// Mitsubishi GX Works2 project: PLC   PLC: FX3G

// global labels: Global1
VAR_GLOBAL
  Start_Day AT X007 : BOOL;
  Emergency_Switch AT X005 : BOOL;
  Work_Day AT Y007 : BOOL;
  Y7coil AT Y007 : BOOL;
  MoveInput AT X007 : BOOL;
  RaspInput AT D1100 : REAL;
  RaspInventory AT D1110 : REAL;
  LemonInput AT D1102 : REAL;
  LemonInventory AT D1112 : REAL;
  StabilizerInput AT D1104 : REAL;
  StabilizerInventory AT D1114 : REAL;
  GummyBearsInput AT D1106 : REAL;
  GummyBearsInventory AT D1116 : REAL;
  ReadyGummyGumPackage AT D1108 : REAL;
  Start_Making AT X001 : BOOL;
  Analog_Input AT D8280 : INT;
  Analog_Float AT D8280 : REAL;
END_VAR
VAR_GLOBAL CONSTANT
  Div400 : REAL := 400;
END_VAR
VAR_GLOBAL
  GummyChoice AT D7000 : REAL;
END_VAR
VAR_GLOBAL CONSTANT
  Plesure : REAL := 6;
END_VAR
VAR_GLOBAL
  Pleasure_Check AT M0 : BOOL;
END_VAR
VAR_GLOBAL CONSTANT
  Regular : REAL := 5;
END_VAR
VAR_GLOBAL
  Regular_Check AT M1 : BOOL;
END_VAR
VAR_GLOBAL CONSTANT
  MinRasp : REAL := 385;
  MinLemon : REAL := 455;
END_VAR
VAR_GLOBAL
  CheckLemonRegular AT M23 : BOOL;
END_VAR
VAR_GLOBAL CONSTANT
  StabilizerMin : REAL := 105;
END_VAR
VAR_GLOBAL
  CheckStabilizerReg AT M24 : BOOL;
END_VAR
VAR_GLOBAL CONSTANT
  GummyBearsMin : REAL := 28;
END_VAR
VAR_GLOBAL
  CheckGummyBearsReg AT M25 : BOOL;
  YesRegularInv AT M16 : BOOL;
END_VAR
VAR_GLOBAL CONSTANT
  MinRaspReg : REAL := 280;
  MinLemonReg : REAL := 455;
  StabilizerMinReg : REAL := 105;
  GummyBearsMinReg : REAL := 28;
  MinRaspPleas : REAL := 385;
END_VAR
VAR_GLOBAL
  CheckRaspPleas AT M26 : BOOL;
END_VAR
VAR_GLOBAL CONSTANT
  MinLemonPleas : REAL := 665;
END_VAR
VAR_GLOBAL
  CheckLemonPleas AT M27 : BOOL;
END_VAR
VAR_GLOBAL CONSTANT
  StabilizerMinPleas : REAL := 210;
END_VAR
VAR_GLOBAL
  CheckStabilizerPleas AT M28 : BOOL;
END_VAR
VAR_GLOBAL CONSTANT
  GummyBearsMinPleas : REAL := 70;
END_VAR
VAR_GLOBAL
  CheckGummyBearsPleas AT M29 : BOOL;
  CheckRaspReg AT M22 : BOOL;
  YesPleasInv AT M17 : BOOL;
  LackMaterials AT M19 : BOOL;
  IceCreamTimer AT TC1 : BOOL;
END_VAR
VAR_GLOBAL CONSTANT
  IceCreamReady : INT := 50;
END_VAR
VAR_GLOBAL
  InMaking AT TS1 : BOOL;
  MakingProcess AT Y000 : BOOL;
  InMakingProcess AT Y000 : BOOL;
  Start_Cooling AT X002 : BOOL;
  EndMaking AT TS1 : BOOL;
  IceCreamCoolingTimer AT TC2 : BOOL;
END_VAR
VAR_GLOBAL CONSTANT
  IceCreamCool : INT := 80;
END_VAR
VAR_GLOBAL
  InCooling AT TS2 : BOOL;
  TempSens AT X003 : BOOL;
  InCoolingProcess AT Y002 : BOOL;
  Below10Degrees AT X003 : BOOL;
  After8Seconds AT TS2 : BOOL;
  FinishCooloing AT M100 : BOOL;
  gsfg AT M120 : BOOL;
  EndCooking AT TS1 : BOOL;
  FlagEndMaking AT M100 : BOOL;
  RaspIceCreamMaking AT D1210 : REAL;
END_VAR
VAR_GLOBAL CONSTANT
  StabilizerRaspPleas : REAL := 70;
  LemonForRaspPleas : REAL := 105;
END_VAR
VAR_GLOBAL
  LemonIceCreamMaking AT D1212 : REAL;
END_VAR
VAR_GLOBAL CONSTANT
  LemonForLemonPleas : REAL := 560;
  StabilizerLemonPleas : REAL := 140;
  LemonForRaspReg : REAL := 35;
  StabilizeForRaspReg : REAL := 35;
  LemonForLemonReg : REAL := 420;
  StabilzerForLemonReg : REAL := 70;
END_VAR
VAR_GLOBAL
  FlagEndCooling AT M101 : BOOL;
  RaspIceCreamCooling AT D1310 : REAL;
  LemonIceCreamCooling AT D1312 : REAL;
  TimeOfFlicker AT TC3 : BOOL;
END_VAR
VAR_GLOBAL CONSTANT
  FlickeringTimeForPleasure : REAL := 50;
  PleasureFlickeringTime : INT := 50;
END_VAR
VAR_GLOBAL
  TimeOfFlickerRegular AT TC4 : BOOL;
  TimeOfFlickePleas AT TC3 : BOOL;
END_VAR
VAR_GLOBAL CONSTANT
  RegularFlickeringTime : INT := 30;
END_VAR
VAR_GLOBAL
  FlickeringPleas AT TS3 : BOOL;
  FlickeringReg AT TS4 : BOOL;
  MixingContainer AT D1410 : REAL;
  FlickeringHelp AT M10 : BOOL;
  FlickeringLight5IsOver AT TS5 : BOOL;
  BlinkingLight1 AT TC5 : BOOL;
  Light5 AT Y005 : BOOL;
  FlickeringLight2 AT TC6 : BOOL;
  FlickeringLight1 AT TC5 : BOOL;
END_VAR
VAR_GLOBAL CONSTANT
  HalfSecondDuration : INT := 5;
END_VAR
VAR_GLOBAL
  Light6 AT Y006 : BOOL;
  FlickeringLight6IsOver AT TS6 : BOOL;
  StartPackPhase AT X004 : BOOL;
  DonePackage AT CS2 : BOOL;
  PackIceCream AT X000 : BOOL;
  EndPleasureFlickering AT TS3 : BOOL;
  EndRegularFlickering AT TS4 : BOOL;
  FlagEndMixing AT M102 : BOOL;
  ConesCounter AT CC1 : BOOL;
END_VAR
VAR_GLOBAL CONSTANT
  Target : INT := 7;
END_VAR
VAR_GLOBAL
  IceCreamCounter AT CC1 : BOOL;
  FinishPackPhase AT CS1 : BOOL;
  IceCreamCurrentCounter AT CN1 : INT;
END_VAR
VAR_GLOBAL CONSTANT
  Min_For_Y4_Light : INT := 1;
  Max_For_Y4_Light : INT := 6;
END_VAR
VAR_GLOBAL
  Light4 AT Y004 : BOOL;
END_VAR
VAR_GLOBAL CONSTANT
  AddPackage : REAL := 1;
END_VAR
VAR_GLOBAL
  ResetDelay AT TC7 : BOOL;
END_VAR
VAR_GLOBAL CONSTANT
  DelayDuration : INT := 10;
END_VAR
VAR_GLOBAL
  ResetDelayOver AT TS7 : BOOL;
  EndDayReset AT M110 : BOOL;
END_VAR
VAR_GLOBAL CONSTANT
  Normalization : REAL := 40;
END_VAR
VAR_GLOBAL
  NormalizedNumberOfPackages AT D1500 : REAL;
  AnalogOutput AT D8282 : INT;
END_VAR
VAR_GLOBAL CONSTANT
  IngredientsForPleasure : REAL := 190;
  IngredientsForRegular : REAL := 124;
END_VAR
VAR_GLOBAL
  EndIteration AT M200 : BOOL;
END_VAR

// task Task_01 (event TRUE, interval 0, priority 31): POU_01

PROGRAM POU_01
VAR
  CheckRaspRegular : BOOL;
END_VAR
(* structured ladder/FBD written out as ST: instructions are called as NAME(EN, inputs, outputs); _pN, _eN, _tN stand for wires *)
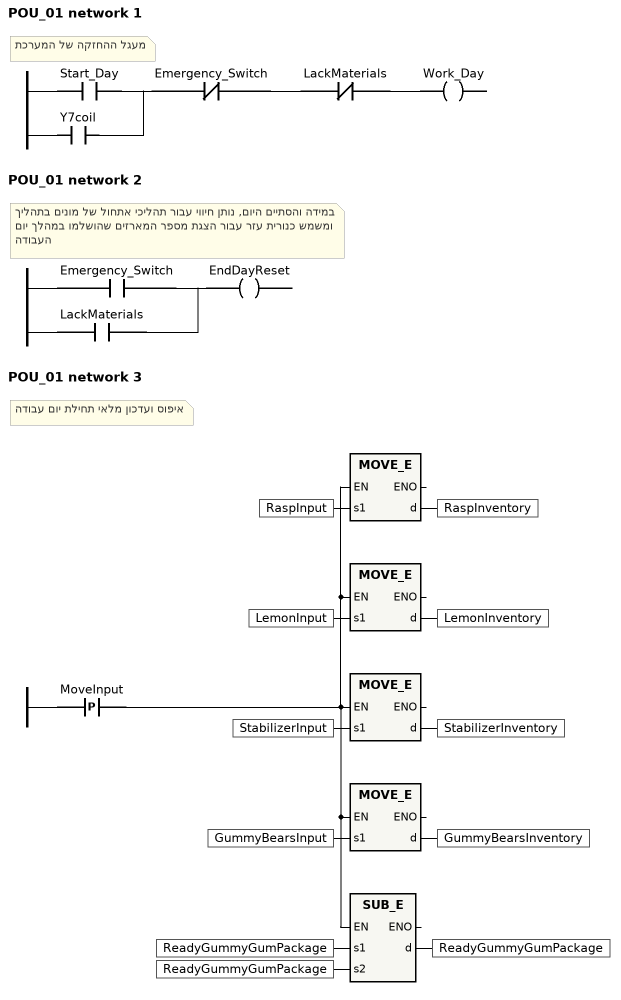
(* network 1 *)
(* מעגל ההחזקה של המערכת *)
Work_Day := ((Start_Day OR Y7coil) AND NOT Emergency_Switch) AND NOT LackMaterials;
(* network 2 *)
(* במידה והסתיים היום, נותן חיווי עבור תהליכי אתחול של מונים בתהליך ומשמש כנורית עזר עבור הצגת מספר המארזים שהושלמו במהלך יום העבודה *)
EndDayReset := Emergency_Switch OR LackMaterials;
(* network 3 *)
(* איפוס ועדכון מלאי תחילת יום עבודה *)
_p1 := LDP(TRUE, MoveInput);
MOVE_E(_p1, RaspInput, RaspInventory);
MOVE_E(_p1, LemonInput, LemonInventory);
MOVE_E(_p1, StabilizerInput, StabilizerInventory);
MOVE_E(_p1, GummyBearsInput, GummyBearsInventory);
SUB_E(_p1, ReadyGummyGumPackage, ReadyGummyGumPackage, ReadyGummyGumPackage);
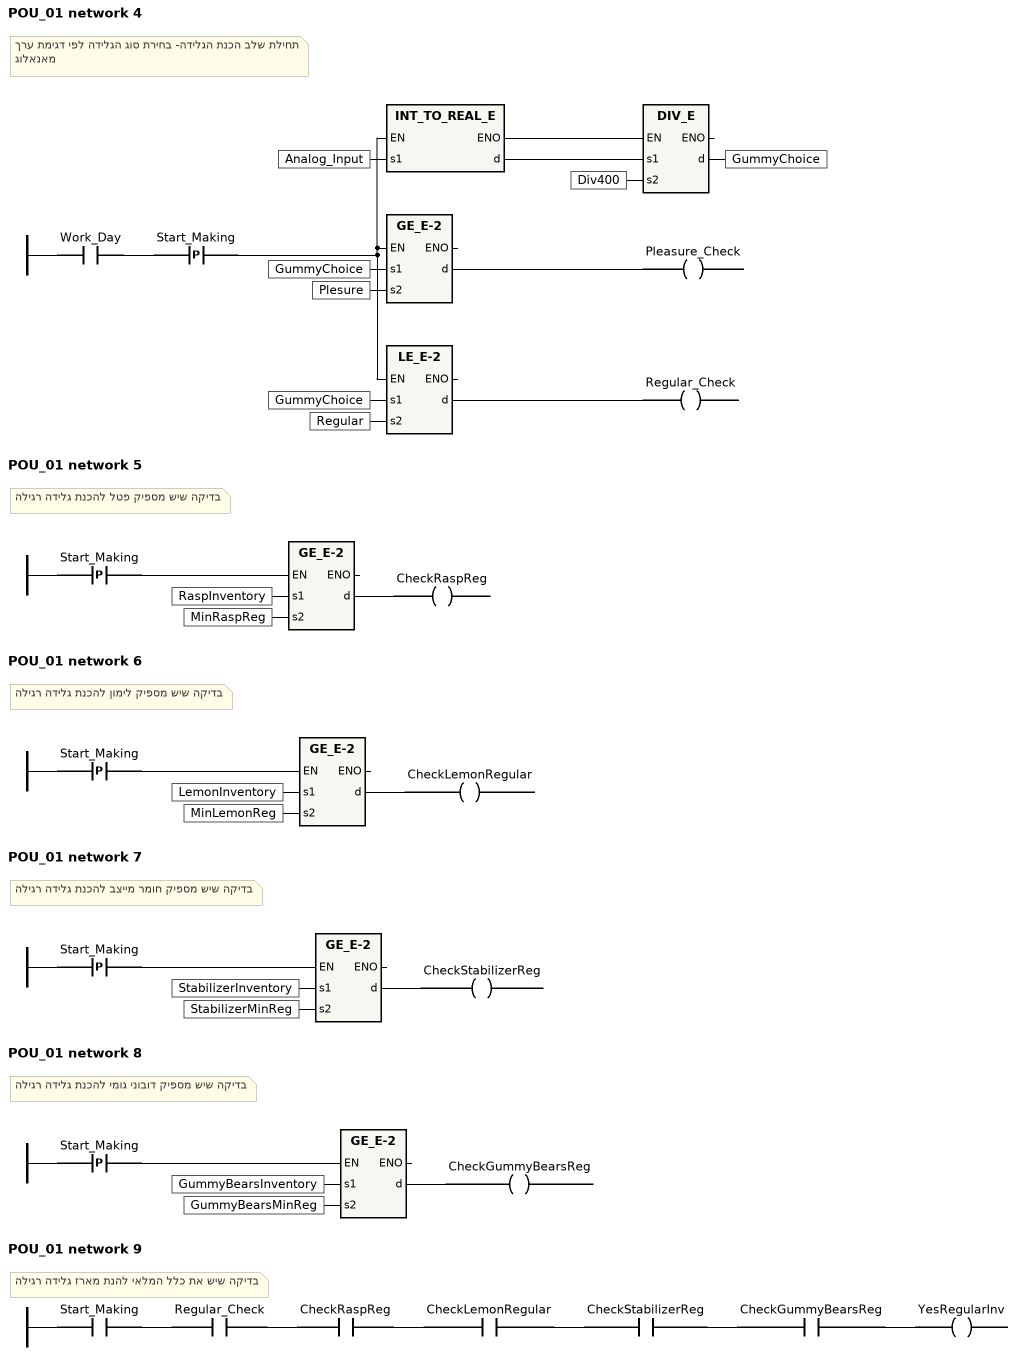
(* network 4 *)
(* תחילת שלב הכנת הגלידה- בחירת סוג הגלידה לפי דגימת ערך מאנאלוג *)
_p1 := Work_Day AND LDP(TRUE, Start_Making);
_e3 := INT_TO_REAL_E(_p1, Analog_Input, _t2);
DIV_E(_e3, _t2, Div400, GummyChoice);
GE_E(_p1, GummyChoice, Plesure, _t4);
Pleasure_Check := _t4;
LE_E(_p1, GummyChoice, Regular, _t5);
Regular_Check := _t5;
(* network 5 *)
(* בדיקה שיש מספיק פטל להכנת גלידה רגילה *)
GE_E(LDP(TRUE, Start_Making), RaspInventory, MinRaspReg, _t1);
CheckRaspReg := _t1;
(* network 6 *)
(* בדיקה שיש מספיק לימון להכנת גלידה רגילה *)
GE_E(LDP(TRUE, Start_Making), LemonInventory, MinLemonReg, _t1);
CheckLemonRegular := _t1;
(* network 7 *)
(* בדיקה שיש מספיק חומר מייצב להכנת גלידה רגילה *)
GE_E(LDP(TRUE, Start_Making), StabilizerInventory, StabilizerMinReg, _t1);
CheckStabilizerReg := _t1;
(* network 8 *)
(* בדיקה שיש מספיק דובוני גומי להכנת גלידה רגילה *)
GE_E(LDP(TRUE, Start_Making), GummyBearsInventory, GummyBearsMinReg, _t1);
CheckGummyBearsReg := _t1;
(* network 9 *)
(* בדיקה שיש את כלל המלאי להנת מארז גלידה רגילה *)
YesRegularInv := Start_Making AND Regular_Check AND CheckRaspReg AND CheckLemonRegular AND CheckStabilizerReg AND CheckGummyBearsReg;
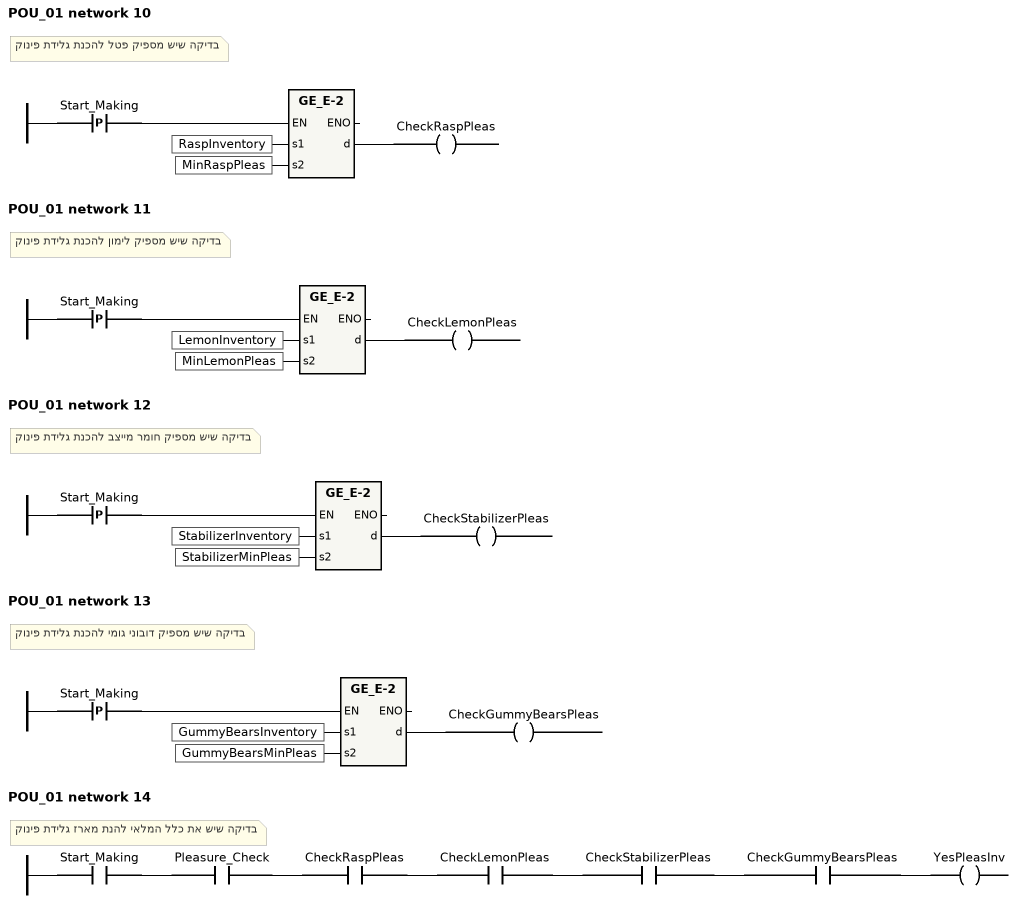
(* network 10 *)
(* בדיקה שיש מספיק פטל להכנת גלידת פינוק *)
GE_E(LDP(TRUE, Start_Making), RaspInventory, MinRaspPleas, _t1);
CheckRaspPleas := _t1;
(* network 11 *)
(* בדיקה שיש מספיק לימון להכנת גלידת פינוק *)
GE_E(LDP(TRUE, Start_Making), LemonInventory, MinLemonPleas, _t1);
CheckLemonPleas := _t1;
(* network 12 *)
(* בדיקה שיש מספיק חומר מייצב להכנת גלידת פינוק *)
GE_E(LDP(TRUE, Start_Making), StabilizerInventory, StabilizerMinPleas, _t1);
CheckStabilizerPleas := _t1;
(* network 13 *)
(* בדיקה שיש מספיק דובוני גומי להכנת גלידת פינוק *)
GE_E(LDP(TRUE, Start_Making), GummyBearsInventory, GummyBearsMinPleas, _t1);
CheckGummyBearsPleas := _t1;
(* network 14 *)
(* בדיקה שיש את כלל המלאי להנת מארז גלידת פינוק *)
YesPleasInv := Start_Making AND Pleasure_Check AND CheckRaspPleas AND CheckLemonPleas AND CheckStabilizerPleas AND CheckGummyBearsPleas;
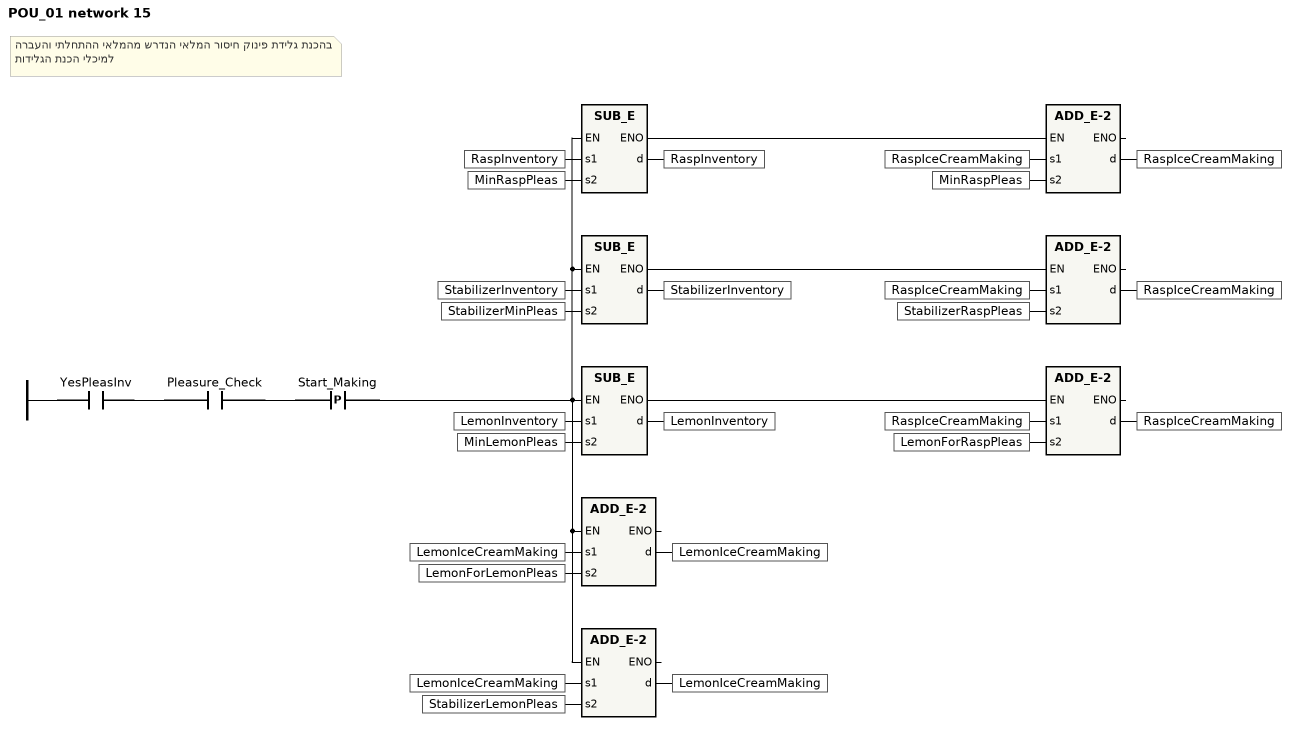
(* network 15 *)
(* בהכנת גלידת פינוק חיסור המלאי הנדרש מהמלאי ההתחלתי והעברה למיכלי הכנת הגלידות *)
_p1 := YesPleasInv AND Pleasure_Check AND LDP(TRUE, Start_Making);
_e2 := SUB_E(_p1, RaspInventory, MinRaspPleas, RaspInventory);
ADD_E(_e2, RaspIceCreamMaking, MinRaspPleas, RaspIceCreamMaking);
_e3 := SUB_E(_p1, StabilizerInventory, StabilizerMinPleas, StabilizerInventory);
ADD_E(_e3, RaspIceCreamMaking, StabilizerRaspPleas, RaspIceCreamMaking);
_e4 := SUB_E(_p1, LemonInventory, MinLemonPleas, LemonInventory);
ADD_E(_e4, RaspIceCreamMaking, LemonForRaspPleas, RaspIceCreamMaking);
ADD_E(_p1, LemonIceCreamMaking, LemonForLemonPleas, LemonIceCreamMaking);
ADD_E(_p1, LemonIceCreamMaking, StabilizerLemonPleas, LemonIceCreamMaking);
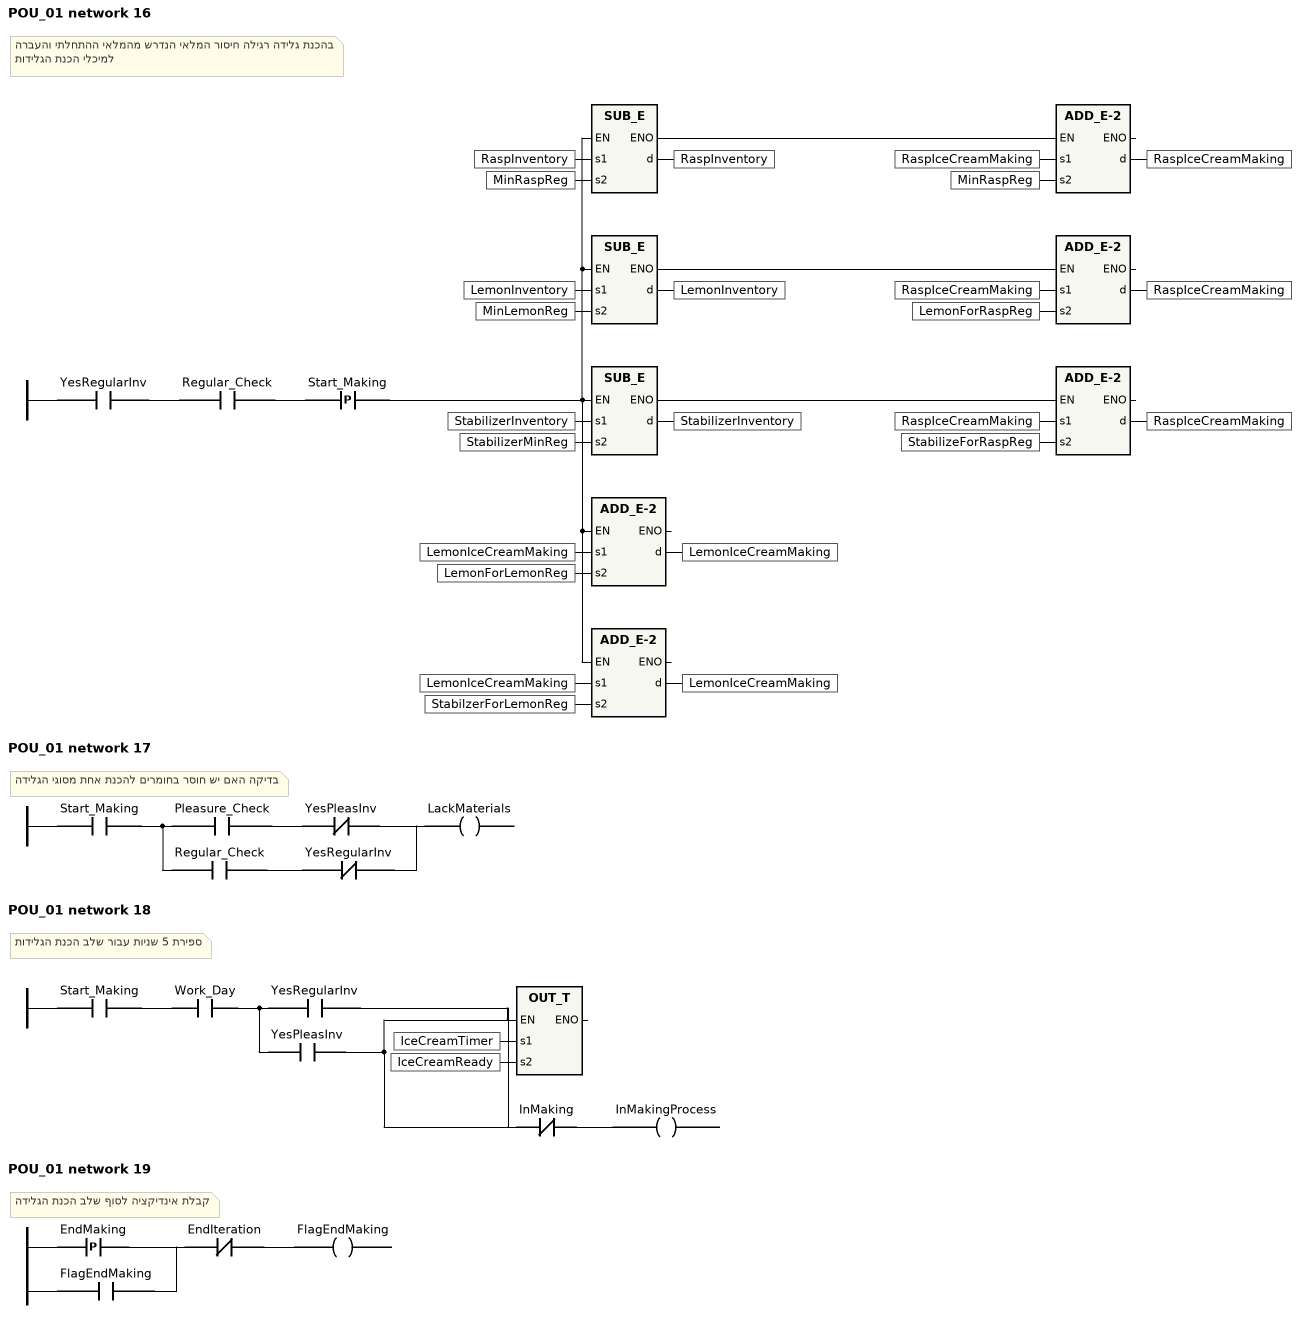
(* network 16 *)
(* בהכנת גלידה רגילה חיסור המלאי הנדרש מהמלאי ההתחלתי והעברה למיכלי הכנת הגלידות *)
_p1 := YesRegularInv AND Regular_Check AND LDP(TRUE, Start_Making);
_e2 := SUB_E(_p1, RaspInventory, MinRaspReg, RaspInventory);
ADD_E(_e2, RaspIceCreamMaking, MinRaspReg, RaspIceCreamMaking);
_e3 := SUB_E(_p1, LemonInventory, MinLemonReg, LemonInventory);
ADD_E(_e3, RaspIceCreamMaking, LemonForRaspReg, RaspIceCreamMaking);
_e4 := SUB_E(_p1, StabilizerInventory, StabilizerMinReg, StabilizerInventory);
ADD_E(_e4, RaspIceCreamMaking, StabilizeForRaspReg, RaspIceCreamMaking);
ADD_E(_p1, LemonIceCreamMaking, LemonForLemonReg, LemonIceCreamMaking);
ADD_E(_p1, LemonIceCreamMaking, StabilzerForLemonReg, LemonIceCreamMaking);
(* network 17 *)
(* בדיקה האם יש חוסר בחומרים להכנת אחת מסוגי הגלידה *)
LackMaterials := (Start_Making AND Pleasure_Check AND NOT YesPleasInv) OR (Start_Making AND Regular_Check AND NOT YesRegularInv);
(* network 18 *)
(* ספירת 5 שניות עבור שלב הכנת הגלידות *)
_p1 := Start_Making AND Work_Day;
_p2 := (_p1 AND YesRegularInv) OR (_p1 AND YesPleasInv);
InMakingProcess := _p2 AND NOT InMaking;
OUT_T(_p2, IceCreamTimer, IceCreamReady);
(* network 19 *)
(* קבלת אינדיקציה לסוף שלב הכנת הגלידה *)
FlagEndMaking := (LDP(TRUE, EndMaking) OR FlagEndMaking) AND NOT EndIteration;
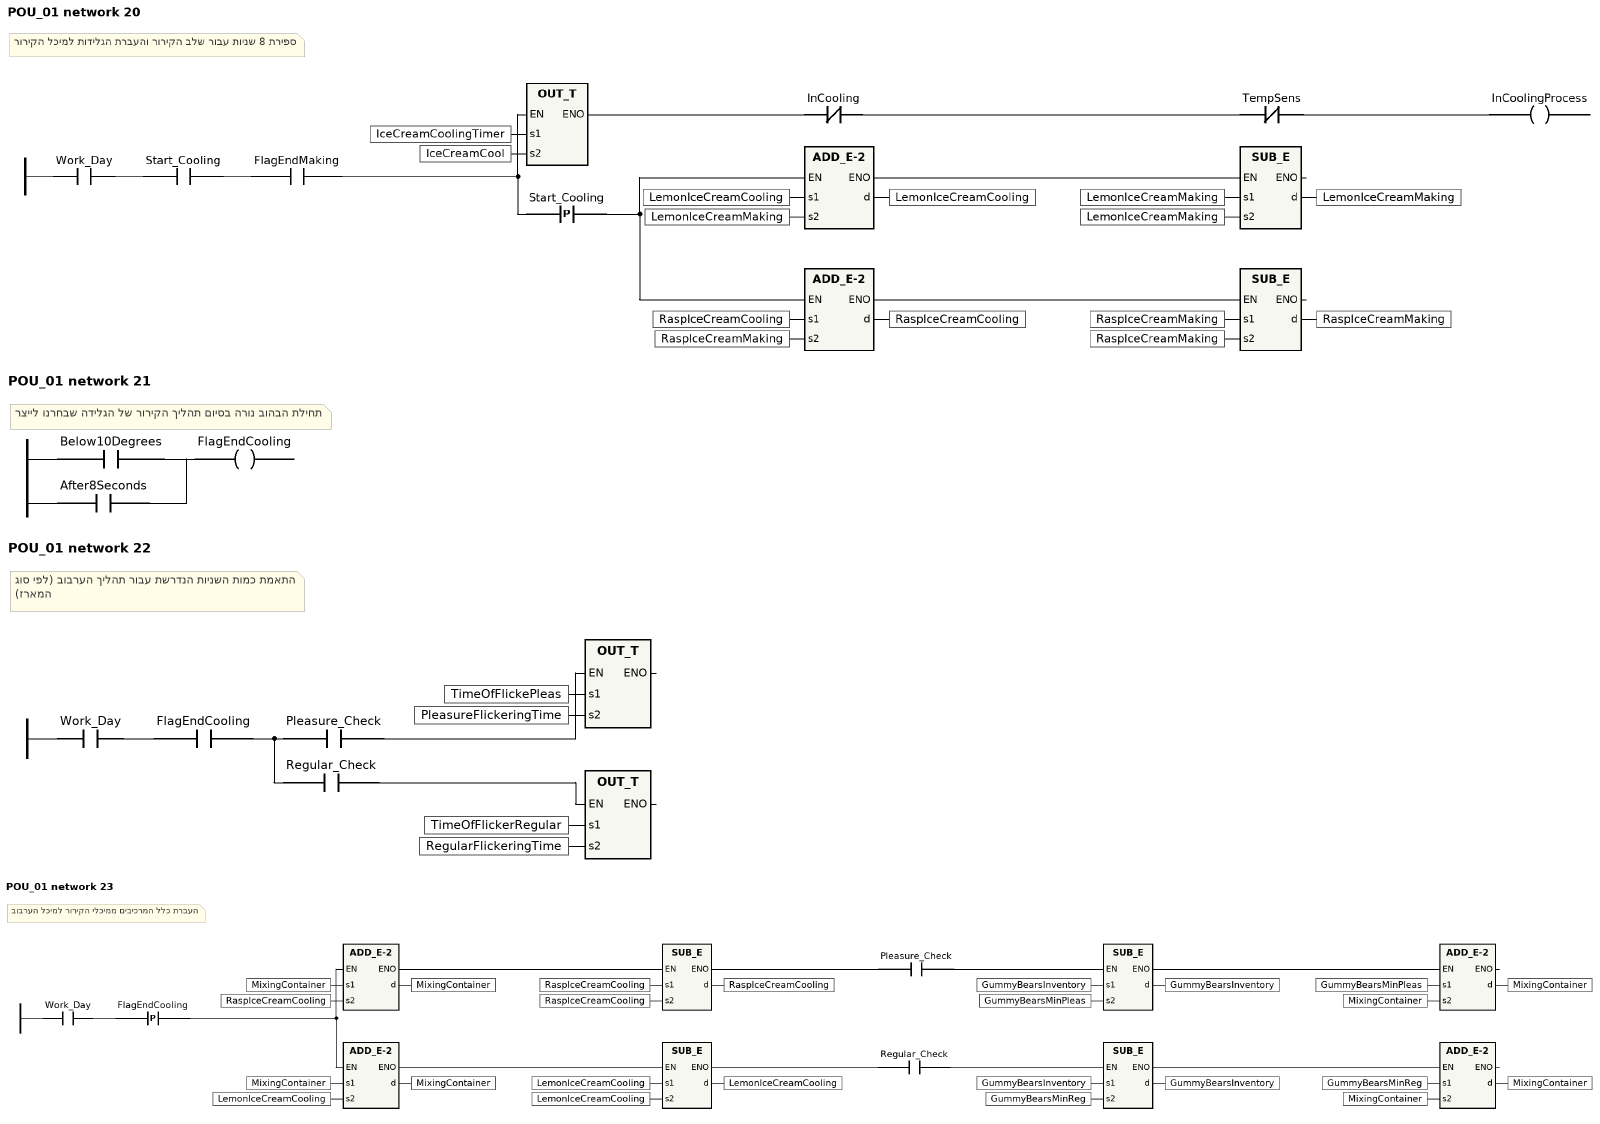
(* network 20 *)
(* ספירת 8 שניות עבור שלב הקירור והעברת הגלידות למיכל הקירור *)
_p1 := Work_Day AND Start_Cooling AND FlagEndMaking;
_e2 := OUT_T(_p1, IceCreamCoolingTimer, IceCreamCool);
InCoolingProcess := _e2 AND NOT InCooling AND NOT TempSens;
_p3 := _p1 AND LDP(TRUE, Start_Cooling);
_e4 := ADD_E(_p3, LemonIceCreamCooling, LemonIceCreamMaking, LemonIceCreamCooling);
SUB_E(_e4, LemonIceCreamMaking, LemonIceCreamMaking, LemonIceCreamMaking);
_e5 := ADD_E(_p3, RaspIceCreamCooling, RaspIceCreamMaking, RaspIceCreamCooling);
SUB_E(_e5, RaspIceCreamMaking, RaspIceCreamMaking, RaspIceCreamMaking);
(* network 21 *)
(* תחילת הבהוב נורה בסיום תהליך הקירור של הגלידה שבחרנו לייצר *)
FlagEndCooling := Below10Degrees OR After8Seconds;
(* network 22 *)
(* התאמת כמות השניות הנדרשת עבור תהליך הערבוב (לפי סוג המארז) *)
_p1 := Work_Day AND FlagEndCooling;
OUT_T(_p1 AND Pleasure_Check, TimeOfFlickePleas, PleasureFlickeringTime);
OUT_T(_p1 AND Regular_Check, TimeOfFlickerRegular, RegularFlickeringTime);
(* network 23 *)
(* העברת כלל המרכיבים ממיכלי הקירור למיכל הערבוב *)
_p1 := Work_Day AND LDP(TRUE, FlagEndCooling);
_e2 := ADD_E(_p1, MixingContainer, RaspIceCreamCooling, MixingContainer);
_e3 := SUB_E(_e2, RaspIceCreamCooling, RaspIceCreamCooling, RaspIceCreamCooling);
_e4 := SUB_E(_e3 AND Pleasure_Check, GummyBearsInventory, GummyBearsMinPleas, GummyBearsInventory);
ADD_E(_e4, GummyBearsMinPleas, MixingContainer, MixingContainer);
_e5 := ADD_E(_p1, MixingContainer, LemonIceCreamCooling, MixingContainer);
_e6 := SUB_E(_e5, LemonIceCreamCooling, LemonIceCreamCooling, LemonIceCreamCooling);
_e7 := SUB_E(_e6 AND Regular_Check, GummyBearsInventory, GummyBearsMinReg, GummyBearsInventory);
ADD_E(_e7, GummyBearsMinReg, MixingContainer, MixingContainer);
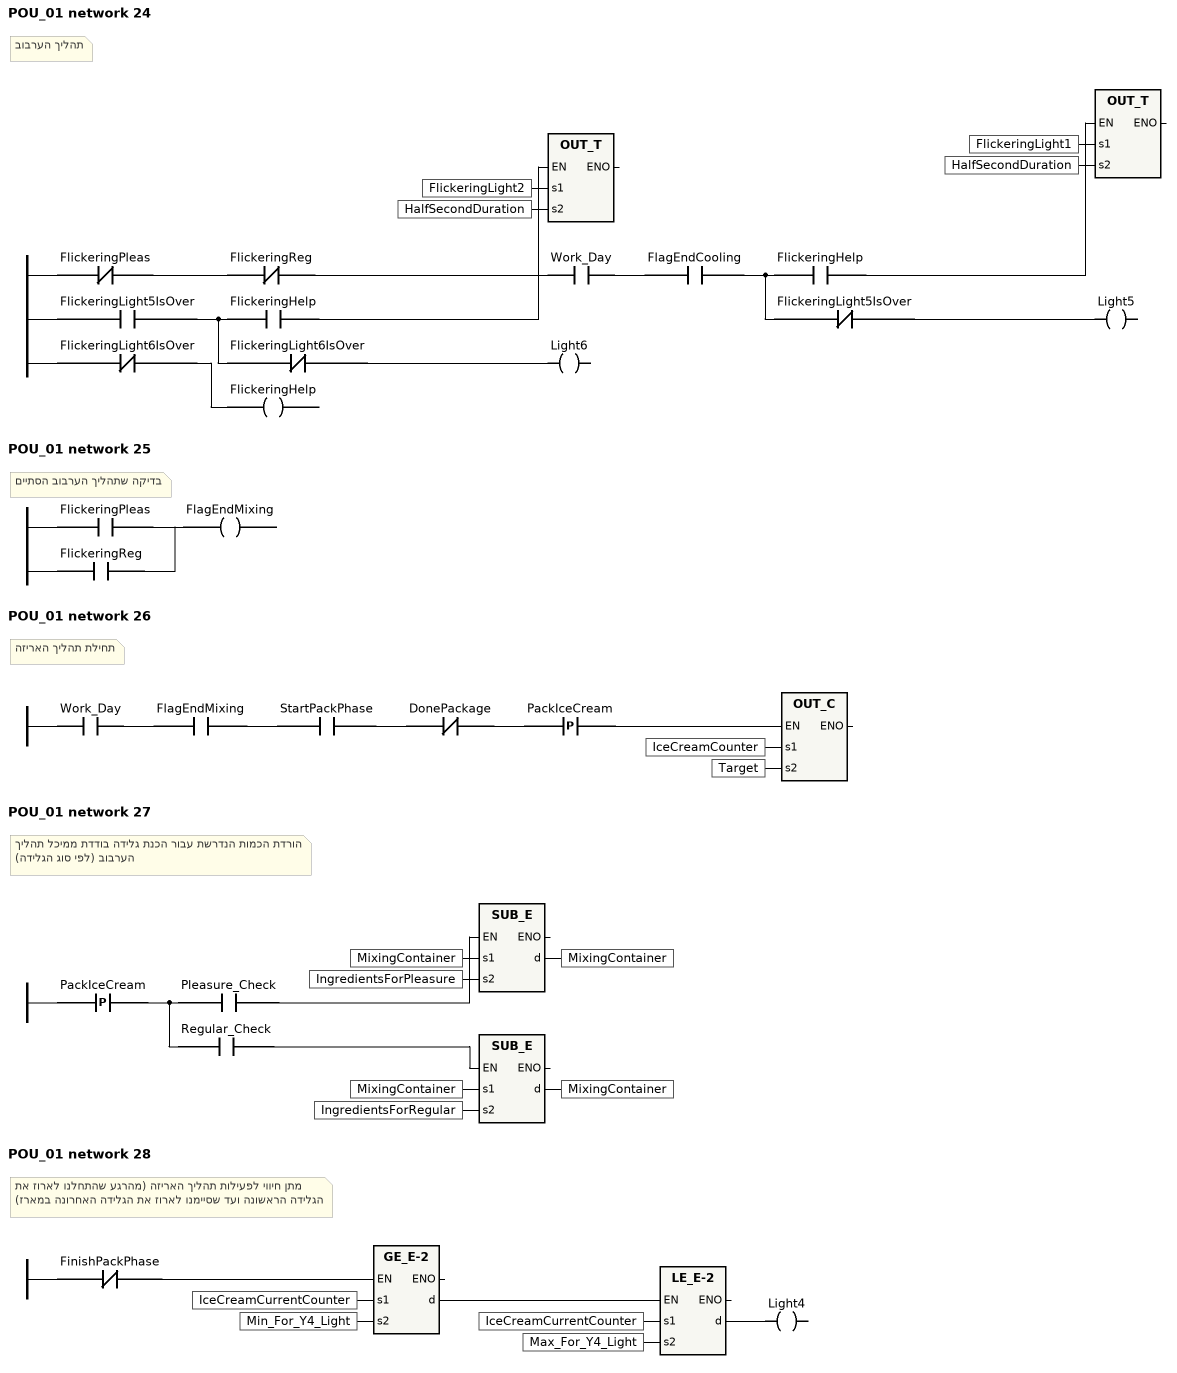
(* network 24 *)
(* תהליך הערבוב *)
_p1 := NOT FlickeringPleas AND NOT FlickeringReg AND Work_Day AND FlagEndCooling;
OUT_T(_p1 AND FlickeringHelp, FlickeringLight1, HalfSecondDuration);
Light5 := _p1 AND NOT FlickeringLight5IsOver;
OUT_T(FlickeringLight5IsOver AND FlickeringHelp, FlickeringLight2, HalfSecondDuration);
Light6 := FlickeringLight5IsOver AND NOT FlickeringLight6IsOver;
FlickeringHelp := NOT FlickeringLight6IsOver;
(* network 25 *)
(* בדיקה שתהליך הערבוב הסתיים *)
FlagEndMixing := FlickeringPleas OR FlickeringReg;
(* network 26 *)
(* תחילת תהליך האריזה *)
OUT_C(Work_Day AND FlagEndMixing AND StartPackPhase AND NOT DonePackage AND LDP(TRUE, PackIceCream), IceCreamCounter, Target);
(* network 27 *)
(* הורדת הכמות הנדרשת עבור הכנת גלידה בודדת ממיכל תהליך הערבוב (לפי סוג הגלידה) *)
_p1 := LDP(TRUE, PackIceCream);
SUB_E(_p1 AND Pleasure_Check, MixingContainer, IngredientsForPleasure, MixingContainer);
SUB_E(_p1 AND Regular_Check, MixingContainer, IngredientsForRegular, MixingContainer);
(* network 28 *)
(* מתן חיווי לפעילות תהליך האריזה (מהרגע שהתחלנו לארוז את הגלידה הראשונה ועד שסיימנו לארוז את הגלידה האחרונה במארז) *)
GE_E(NOT FinishPackPhase, IceCreamCurrentCounter, Min_For_Y4_Light, _t1);
LE_E(_t1, IceCreamCurrentCounter, Max_For_Y4_Light, _t2);
Light4 := _t2;
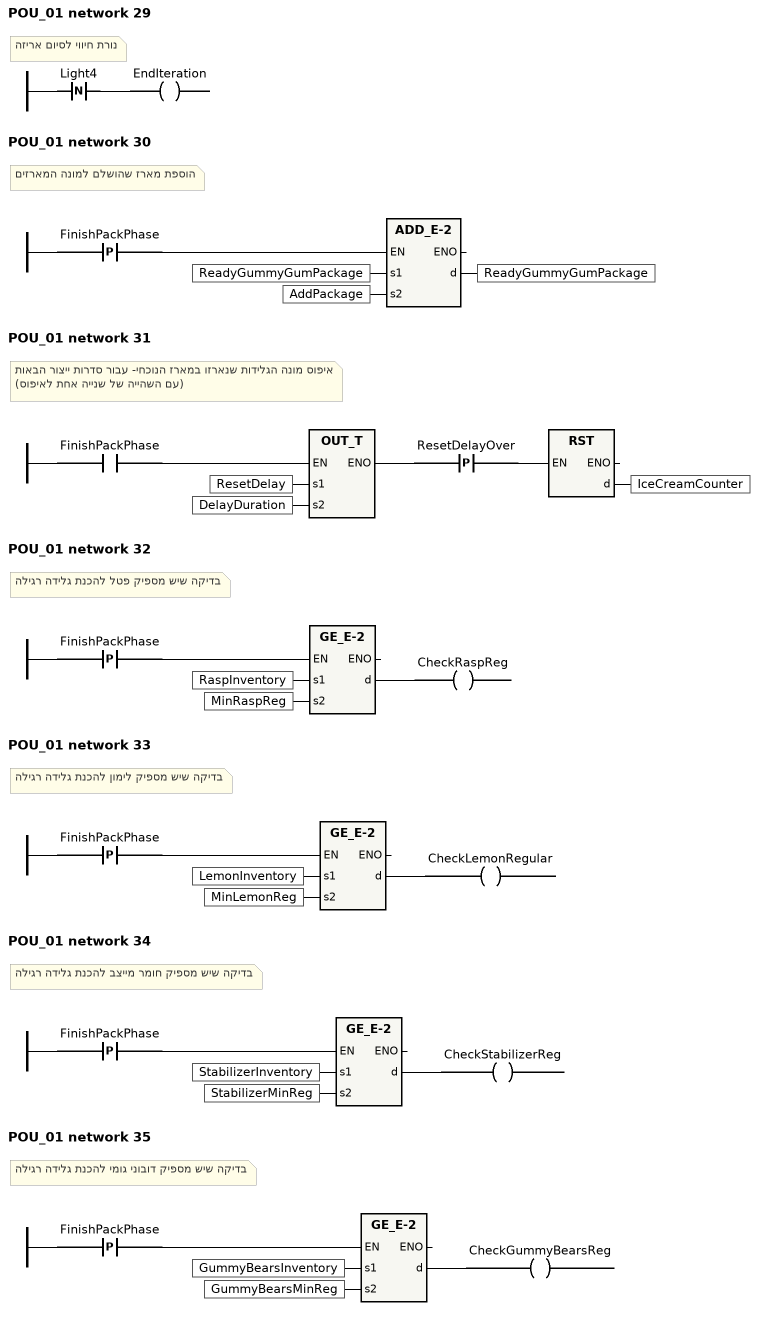
(* network 29 *)
(* נורת חיווי לסיום אריזה *)
EndIteration := LDF(TRUE, Light4);
(* network 30 *)
(* הוספת מארז שהושלם למונה המארזים *)
ADD_E(LDP(TRUE, FinishPackPhase), ReadyGummyGumPackage, AddPackage, ReadyGummyGumPackage);
(* network 31 *)
(* איפוס מונה הגלידות שנארזו במארז הנוכחי- עבור סדרות ייצור הבאות (עם השהייה של שנייה אחת לאיפוס) *)
_e1 := OUT_T(FinishPackPhase, ResetDelay, DelayDuration);
RST(_e1 AND LDP(TRUE, ResetDelayOver), IceCreamCounter);
(* network 32 *)
(* בדיקה שיש מספיק פטל להכנת גלידה רגילה *)
GE_E(LDP(TRUE, FinishPackPhase), RaspInventory, MinRaspReg, _t1);
CheckRaspReg := _t1;
(* network 33 *)
(* בדיקה שיש מספיק לימון להכנת גלידה רגילה *)
GE_E(LDP(TRUE, FinishPackPhase), LemonInventory, MinLemonReg, _t1);
CheckLemonRegular := _t1;
(* network 34 *)
(* בדיקה שיש מספיק חומר מייצב להכנת גלידה רגילה *)
GE_E(LDP(TRUE, FinishPackPhase), StabilizerInventory, StabilizerMinReg, _t1);
CheckStabilizerReg := _t1;
(* network 35 *)
(* בדיקה שיש מספיק דובוני גומי להכנת גלידה רגילה *)
GE_E(LDP(TRUE, FinishPackPhase), GummyBearsInventory, GummyBearsMinReg, _t1);
CheckGummyBearsReg := _t1;
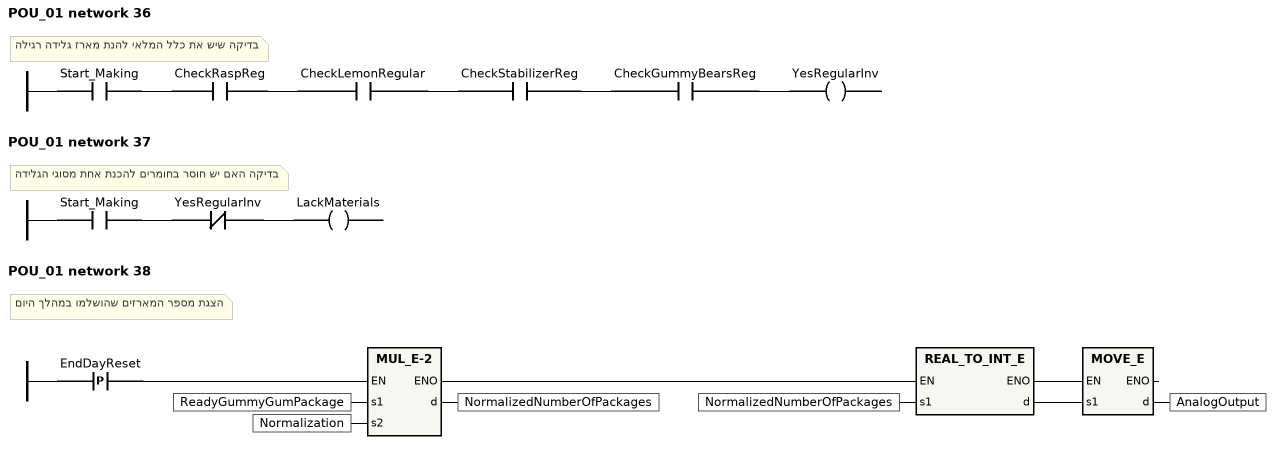
(* network 36 *)
(* בדיקה שיש את כלל המלאי להנת מארז גלידה רגילה *)
YesRegularInv := Start_Making AND CheckRaspReg AND CheckLemonRegular AND CheckStabilizerReg AND CheckGummyBearsReg;
(* network 37 *)
(* בדיקה האם יש חוסר בחומרים להכנת אחת מסוגי הגלידה *)
LackMaterials := Start_Making AND NOT YesRegularInv;
(* network 38 *)
(* הצגת מספר המארזים שהושלמו במהלך היום *)
_e1 := MUL_E(LDP(TRUE, EndDayReset), ReadyGummyGumPackage, Normalization, NormalizedNumberOfPackages);
_e3 := REAL_TO_INT_E(_e1, NormalizedNumberOfPackages, _t2);
MOVE_E(_e3, _t2, AnalogOutput);
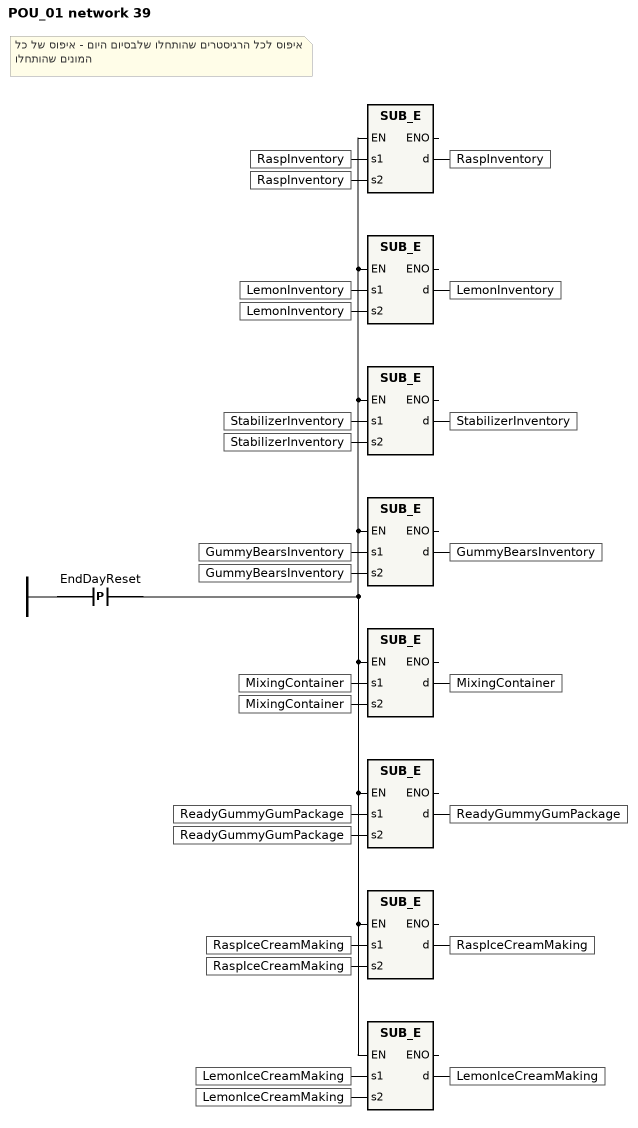
(* network 39 *)
(* איפוס לכל הרגיסטרים שהותחלו שלבסיום היום - איפוס של כל המונים שהותחלו *)
_p1 := LDP(TRUE, EndDayReset);
SUB_E(_p1, RaspInventory, RaspInventory, RaspInventory);
SUB_E(_p1, LemonInventory, LemonInventory, LemonInventory);
SUB_E(_p1, StabilizerInventory, StabilizerInventory, StabilizerInventory);
SUB_E(_p1, GummyBearsInventory, GummyBearsInventory, GummyBearsInventory);
SUB_E(_p1, MixingContainer, MixingContainer, MixingContainer);
SUB_E(_p1, ReadyGummyGumPackage, ReadyGummyGumPackage, ReadyGummyGumPackage);
SUB_E(_p1, RaspIceCreamMaking, RaspIceCreamMaking, RaspIceCreamMaking);
SUB_E(_p1, LemonIceCreamMaking, LemonIceCreamMaking, LemonIceCreamMaking);
END_PROGRAM
